# EPICS substitutions: db/Baumer/ecmcEAM580.substitutions
file "ecmcEAM580-chX.template"
{
  pattern {CH_ID }
          {01    }
}
